{attribute 'GeneratedUsingTerminal: EP4378-1022-0017'}
{attribute addProperty BoxType "EP4378-1022-0017"}
{attribute addProperty Id "Analog_outputAT %Q*INT2"}
{attribute addProperty CRC "3128867708"}
{attribute addProperty Size "2"}
TYPE AO_X06_Pin5_Standard_BA7EBB7C :
STRUCT
	{attribute addProperty Name "Analog_output"}
	Analog_output AT %Q* : INT;
END_STRUCT
END_TYPE

(* stored: Version 1.2.0.0, ProductVersion 3.1.4024.9
   DUT AO_X06_Pin5_Standard_BA7EBB7C: Id {afa23553-c3d3-438b-950a-e055fd5d92d7} *)
